// TIA Portal V18 export
DATA_BLOCK "ST10_GeneralData"   // DB1059
{ S7_Optimized_Access := 'FALSE' }
// stored: AutoNumber false
   VAR
      P_Plus : Array[0..50] of Bool;   // 脉冲沿信号使用Bool,使用需加注释
      ByPass : Array[0..10] of Bool;   // 屏蔽信号,使用需加注释
      HMI : Struct
         AREAPOINTER : Struct
            COORDINATION : Array[1..16] of Bool;
            USER_VERSION : Word;
            SCREEN_NUMBER : Struct
               SCREENTYPE : Int;
               SCREENNUMBER : Int;
               SPARE_1 : Int;
               FIELDNUMBER : Int;
               SPARE_2 : Int;
            END_STRUCT;
            JOB_MAILBOX : Struct
               JOBNUMBER : Int;
               PARAMETER_1 : Int;
               PARAMETER_2 : Int;
               PARAMETER_3 : Int;
            END_STRUCT;
            DATE_TIME_OP : Array[1..12] of Byte;
            DATE_TIME_PLC : Array[1..12] of Byte;
            SPARE : Array[1..22] of Byte;
            DataRecord : Struct   // 数据记录
               RecipeNummer : Word;
               DataRecordNummer : Word;
               Reserve : Word;
               TransferStatus : Word;   // 0,允许传送；2正在传送；4传送已完成，没有错误；12传送完成，出现错误
               Reserve_1 : Word;
            END_STRUCT;
         END_STRUCT;
         Win : Struct   // 弹窗相关变量
            Win : Int;
            WinBullfer : Int;
            "10x弹窗" : Array[1..10] of Int;
            "20x弹窗" : Array[1..10] of Int;
            "30x弹窗" : Array[1..10] of Int;
            "40x弹窗" : Array[1..10] of Int;
            TON : Array[1..40] of TON_TIME;
            "INT" { S7_SetPoint := 'True'} : Array[1..40] of Int;
            "Bool" : Array[1..40] of Bool;
         END_STRUCT;
         StationLightPB : Bool;   // 设备照明按钮
      END_STRUCT;
      Operator : Struct   // 操作员信息
         "Name" : String;   // 姓名
         ID : String;   // 工号
      END_STRUCT;
      TowerLamp : Struct
         PreReady : Bool;   // 等待托盘/等待人工操作
         PreStart : Bool;   // 人工操作完成（自动站False）
         ProcessingFinish : Bool;   // 加工完了 （单个产品加工完成）下个循环开始复位
         Maintenance : Bool;   // 维护提示（缺料OR保养置位1） 无---Flase
      END_STRUCT;
      FlowPartStatus { S7_SetPoint := 'True'} : Array[1..32] of Int;
      FunctionDeSelect : Struct   // 功能屏蔽选择
         "A" : Struct   // 单站屏蔽
            DeSelectPB_Servo380A1 : Bool;
            FunctionDeSelected_Servo380A1 : Bool;
            DeSelectPB_Servo381A1 : Bool;
            FunctionDeSelected_Servo381A1 : Bool;
            DeSelectPB_Servo383A1 : Bool;
            FunctionDeSelected_Servo383A1 : Bool;
            DeSelectPB_Reader800A1 : Bool;
            FunctionDeSelected_Reader800A1 : Bool;
            DeSelectPB_Reader801A1 : Bool;
            FunctionDeSelected_Reader801A1 : Bool;
            DeSelectPB_Reader802A1 : Bool;
            FunctionDeSelected_Reader802A1 : Bool;
            DeSelectPB_Reader803A1 : Bool;
            FunctionDeSelected_Reader803A1 : Bool;
            DeSelectPB_Reader804A1 : Bool;
            FunctionDeSelected_Reader804A1 : Bool;
         END_STRUCT;
         "B" : Struct   // RFID屏蔽
            DeSelectPB_Press372A1 : Bool;
            FunctionDeSelected_Press372A1 : Bool;
            DeSelectPB_Press375A1 : Bool;
            FunctionDeSelected_Press375A1 : Bool;
            DeSelectPB_Reader806A1 : Bool;
            FunctionDeSelected_Reader806A1 : Bool;
            DeSelectPB_TestPress372A1 : Bool;
            FunctionDeSelected_TestPress372A1 : Bool;
            DeSelectPB_TestPress375A1 : Bool;
            FunctionDeSelected_TestPress375A1 : Bool;
         END_STRUCT;
         C : Struct   // 扫码枪屏蔽
            DeSelectPB_Servo382A1 : Bool;
            FunctionDeSelected_Servo382A1 : Bool;
            DeSelectPB_ServoIAI : Bool;
            FunctionDeSelected_ServoIAI : Bool;
            DeSelectPB_IV3810A1 : Bool;
            FunctionDeSelected_IV3810A1 : Bool;
            DeSelectPB_IV3811A1 : Bool;
            FunctionDeSelected_IV3811A1 : Bool;
            DeSelectPB_Glue : Bool;
            FunctionDeSelected_Glue : Bool;
         END_STRUCT;
         "E" : Struct   // 注油屏蔽
            DeSelectPB : Bool;
            FunctionDeSelected : Bool;
         END_STRUCT;
         F : Struct   // 螺丝枪屏蔽
            DeSelectPB_Reader805A1 : Bool;
            FunctionDeSelected_Reader805A1 : Bool;
         END_STRUCT;
         H : Struct   // 油漆笔屏蔽
            DeSelectPB : Bool;
            FunctionDeSelected : Bool;
         END_STRUCT;
         J : Struct   // 油漆笔屏蔽
            DeSelectPB : Bool;
            FunctionDeSelected : Bool;
         END_STRUCT;
         K : Struct   // 油漆笔屏蔽
            DeSelectPB : Bool;
            FunctionDeSelected : Bool;
         END_STRUCT;
         L : Struct   // 油漆笔屏蔽
            DeSelectPB : Bool;
            FunctionDeSelected : Bool;
         END_STRUCT;
         MES : Struct   // MES屏蔽
            DeSelectPB : Bool;
            FunctionDeSelected : Bool;
         END_STRUCT;
         Global : Struct
            DeSelectPB_DryMode : Bool;
            FunctionDeSelected_DryMode : Bool;
            DeSelectPB_ScanFixture : Bool;
            FunctionDeSelected_ScanFixture : Bool;
            Spare_2 : Bool;
            Spare_3 : Bool;
            Spare_4 : Bool;
            Spare_5 : Bool;
            Spare_6 : Bool;
            Spare_7 : Bool;
            Spare_8 : Bool;
            Spare_9 : Bool;
            Spare_10 : Bool;
            Spare_11 : Bool;
            Spare_12 : Bool;
            Spare_13 : Bool;
         END_STRUCT;
      END_STRUCT;
      FlowControl_Handshake : Array[1..32] of Struct   // 流程控制的互锁
         PartPresent : Bool;
         initi : Bool;   // 初始化
         Start : Bool;
         Running : Bool;
         Done : Bool;
         Bypass : Bool;
      END_STRUCT;
      FixtureIDCheck { S7_SetPoint := 'True'} : Array[1..16] of "FixtureCheck_UDT";   // 工装匹配
      ProcessData { S7_SetPoint := 'True'} : Array[0..5] of "ProcessDatad";
   END_VAR
BEGIN
   // FlowControl_Handshake[2].Bypass : 流程NG
   // FlowControl_Handshake[1] : 主加工流程控制的互锁
   // FlowControl_Handshake[2] : 打标流程控制的互锁
   // FlowControl_Handshake[3] : 产品定位流程控制的互锁
   // FlowControl_Handshake[4] : 贴标流程控制互锁
END_DATA_BLOCK
